# EPICS autosave request: iocBoot/iocmmc100test/auto_positions.req
file motor_positions.req P=MLL:,M=sphi
